FUNCTION_BLOCK FB_Basis
VAR_INPUT
END_VAR
VAR_OUTPUT
END_VAR
VAR
	bStart			:BOOL;		// Variable für internes handling der Eigenschaft 
	bStop			:BOOL;		// Variable für internes handling der Eigenschaft 
END_VAR

METHOD M_Start : BOOL
VAR_INPUT
END_VAR
bStart := TRUE;
bStop := FALSE;
END_METHOD

METHOD M_Stop : BOOL
VAR_INPUT
END_VAR
bStart := FALSE;
bStop := TRUE;
END_METHOD

PROPERTY P_State : BOOL
GET
P_State := bStop;
END_GET
END_PROPERTY

END_FUNCTION_BLOCK

(* stored: Version 1.1.0.1
   POU FB_Basis: Id {fffd0907-c1c1-493c-ac2c-314e9089ee0d}, SpecialFunc None
   Method M_Start: Id {814a3d4c-bdf1-4ff2-b4ec-cf40aba645ba}
   Method M_Stop: Id {645c63c8-13f0-478f-ae7b-32e8477e4722}
   Property P_State: Id {ffbbd73b-900a-4aee-bc8d-5f319a8cfba9}
   Get Get: Id {7a5f06a2-1350-4bac-a53f-e294f574a899} *)
